// TIA Portal V18 export
FUNCTION_BLOCK "hour_min"   // FB6, LAD
{ S7_Optimized_Access := 'TRUE' }
VERSION : 0.1
// stored: AutoNumber true, IsIECCheckEnabled false, IsRetainMemResEnabled false, MemoryReserve 100, SetENOAutomatically false, UDAEnableTagReadback false
   VAR_INPUT
      in : Bool;
      reset : Bool;
   END_VAR
   VAR_OUTPUT
      outmin : Int;
      outhr : Int;
   END_VAR
   VAR RETAIN
      insec : Int;
   END_VAR
   VAR
      temp : Bool;
   END_VAR
   VAR_TEMP   // added for the SCL form of the ladder/FBD networks
      _w1 : Bool;
   END_VAR
BEGIN

REGION Network 1
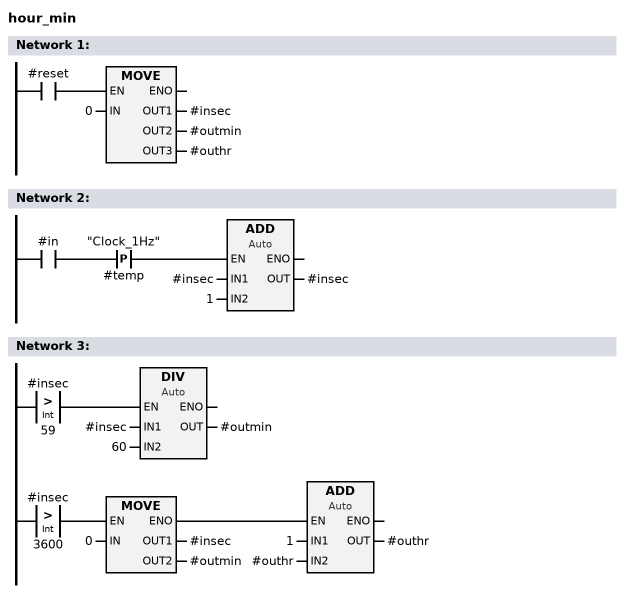
   RUNG wire#powerrail
      Contact( #reset )
      Move(in := 0, out1 => #insec, out2 => #outmin, out3 => #outhr)
   END_RUNG
   // the same network as SCL:
   IF #reset THEN
       #insec := 0;
       #outmin := 0;
       #outhr := 0;
   END_IF;
END_REGION

REGION Network 2
   RUNG wire#powerrail
      Contact( #in )
      P_Contact(operand := "Clock_1Hz", bit := #temp)
      Add(in1 := #insec, in2 := 1, out => #insec)
   END_RUNG
   // the same network as SCL:
   #_w1 := #in AND "Clock_1Hz" AND NOT #temp;   // rising edge of "Clock_1Hz"
   #temp := "Clock_1Hz";
   IF #_w1 THEN #insec := #insec + 1; END_IF;
END_REGION

REGION Network 3
   RUNG wire#powerrail
      { S7_Templates := "SrcType := Int" } GT_Contact(in1 := #insec, in2 := 59)
      Div(in1 := #insec, in2 := 60, out => #outmin)
   END_RUNG
   RUNG wire#powerrail
      { S7_Templates := "SrcType := Int" } GT_Contact(in1 := #insec, in2 := 3600)
      Move(in := 0, out1 => #insec, out2 => #outmin)
      Add(in1 := 1, in2 := #outhr, out => #outhr)
   END_RUNG
   // the same network as SCL:
   IF #insec > 59 THEN #outmin := #insec / 60; END_IF;
   #_w1 := #insec > 3600;
   IF #_w1 THEN
       #insec := 0;
       #outmin := 0;
       #outhr := 1 + #outhr;
   END_IF;
END_REGION
END_FUNCTION_BLOCK
